(* CODESYS project Sample20190212.project

Project tree, tasks and I/O mapping:
  Device : Changsha-Cyber-MI-linux, Changsha Cyber-MI Co., Ltd., version 3.5.10.40
    application Application
      libraries: Standard, * (System); CANbus, 3.5.7.0 (3S - Smart Software Solutions GmbH); SysMem, 3.5.12.0 (System); CAA SerialCom, 3.5.12.0 (CAA Technical Workgroup); CAA Net Base Services, 3.5.12.0 (CAA Technical Workgroup); cyber gpio, 3.5.10.40 (cyber); cyber udp lib , 3.5.10.41 (cyber Inc.); SysTypes2 Interfaces, 3.5.4.0 (System); SysFile, 3.5.9.0 (System); VisuDialogs, * (System)
      task MainTask (cyclic, interval 4 ms, priority 1) calls prg_running
      task Task_running (cyclic, interval 10 ms, priority 1) calls prg_button
      task Task_CAN0 (cyclic, interval 50 ms, priority 1) calls prg_can0
      task Task_RS485 (cyclic, interval 50 ms, priority 1) calls COM_SERIAL
      task Task_Ethernet (cyclic, interval t#20ms, priority 1) calls Ethernet
      task Task_falsecheck (cyclic, interval t#20ms, priority 1) calls FaultCheck
      task Task_GPRS (cyclic, interval t#20ms, priority 1) calls GPRS
      task Task_files (cyclic, interval t#20ms, priority 1) calls Files
      task VISU_TASK (cyclic, interval 100 ms, priority 31) calls VisuElems.Visu_Prg
      CAN0/
        program prg_can0 [ST]
        function CAN_Send_MSG [ST]
      DI_DO/
        program prg_running [ST]
        program prg_button [ST]
      global variables GVL
      RS485/
        program COM_SERIAL [ST]
      Ethernet/
        data type STATE
        program Ethernet [ST]
      FaultCheck/
        function block FB_Fault [ST]
        program FaultCheck [ST]
      GPRS/
        program GPRS [ST]
      Files/
        program Files [ST]
      visualisation Visualization_files
    SoftMotion General Axis Pool
    IoDrvMIC7001 : IoDrvMIC7001, MyCompany, version 18.11.1
        input  Application.GVL.DI_button : BOOL  // Di02-Ai02@C17
        output Application.GVL.DO_running : BOOL  // LED_run
        output Application.GVL.DO_error : BOOL  // LED_err
        unmapped channels: Ai00@C16, Ai01@C28, Ai02@C17, Ai03@C29, Ai04@C30, Ai05@C19, Ai06@C31, Ai07@C20, Ai08@C18, Ai09@D18, Ai10@D20, Ai11@D31, Ai12@D19, Ai13@D30, Ai14@D29, Ai15@D17, Ai16@D28, Ai17@D16, Ai18-Do00@C25, Ai19-Do01@C24, Ai20-Do02@C13, Ai21-Do03@C01, Ai22-Do04@C03, Ai23-Do05@C04, Ai24-Do06@C05, Ai25-Do07@C06, Ai26-Do08@C08, Ai27-Do09@C09, Ai28-Do10@C10, Ai29-Do11@C11, Ai30-Do12@D34, Ai31-Do13@D35, Ai32-Do14@D23, Ai33-Do15@D12, Ai34-Do16@D10, Ai35-Do17@D09, Ai36-Do18@D08, Ai37-Do19@D07, Ai38-Do20@D05, Ai39-Do21@D04,
          Ai40-Do22@D03, Ai41-Do23@D02, Ai42-Do24@C23, Ai43-Do25@C35, Ai44-Do26@D24, Ai45-Do27@D13, Ai46-Ao00@C22, Ai47-Ao01@D14, Ai48_Pi02, Ai49_Out5V, Ai50_VCC, Ai51_VCC_L, Ai52_VCC_R, Ai53_Pwm-i0, Ai54_Pwm-i1, Ai55_Pwm-i2, Ai56_Pwm-i3, Ai57_CPU-T, Ai58_G-x, Ai59_G-y, Ai60_G-z, Ai61-reserved, Ai62-IO-cntr, Ai63-CDS-cntr, Di00-Ai00@C16, Di01-Ai01@C28, Di03-Ai03@C29, Di04-Ai04@C30, Di05-Ai05@C19, Di06-Ai06@C31, Di07-Ai07@C20, Di08-Ai08@C18, Di09-Ai09@D18, Di10-Ai10@D20, Di11-Ai11@D31, Di12-Ai12@D19, Di13-Ai13@D30, Di14-Ai14@D29, Di15-Ai15@D17, Di16-Ai16@D28,
          Di17-Ai17@D16, Di18-Ai18@C25, Di19-Ai19@C24, Di20-Ai20@C13, Di21-Ai21@C01, Di22-Ai22@C03, Di23-Ai23@C04, Di24-Ai24@C05, Di25-Ai25@C06, Di26-Ai26@C08, Di27-Ai27@C09, Di28-Ai28@C10, Di29-Ai29@C11, Di30-Ai30@D34, Di31-Ai31@D35, Di32-Ai32@D23, Di33-Ai33@D12, Di34-Ai34@D10, Di35-Ai35@D09, Di36-Ai36@D08, Di37-Ai37@D07, Di38-Ai38@D05, Di39-Ai39@D04, Di40-Ai40@D03, Di41-Ai41@D02, Di42-Ai42@C23, Di43-Ai43@C35, Di44-Ai44@D24, Di45-Ai45@D13, Di46-Ai46@C22, Di47-Ai47@D14, Di48-Pi00@C15, Di49-Pi01@C14, Di50-Pi02@D22, Di51-Pi03@D21, Di52-reserved, Di53-reserved, Di54-reserved, Di55-reserved, Di56-reserved,
          Di57-reserved, Di58-reserved, Di59-reserved, Di60-reserved, Di61-reserved, Di62-reserved, Di63-reserved, Pi00-Di48@C15, Pi01-Di49@C14, Pi02-Di50@D22, Pi03-Di51@D21, Do00-Ai18@C25, Do01-Ai19@C24, Do02-Ai20@C13, Do03-Ai21@C01, Do04-Ai22@C03, Do05-Ai23@C04, Do06-Ai24@C05, Do07-Ai25@C06, Do08-Ai26@C08, Do09-Ai27@C09, Do10-Ai28@C10, Do11-Ai29@C11, Do12-Ai30@D34, Do13-Ai31@D35, Do14-Ai32@D23, Do15-Ai33@D12, Do16-Ai34@D10, Do17-Ai35@D09, Do18-Ai36@D08, Do19-Ai37@D07, Do20-Ai38@D05, Do21-Ai39@D04, Do22-Ai40@D03, Do23-Ai41@D02, Do24-Ai42@C23, Do25-Ai43@C35, Do26-Ai44@D24, Do27-Ai45@D13, Do28-Pwmi00@C33,
          Do29-Pwmi01@C34, Do30-Pwmi02@D25, Do31-Pwmi03@D26, PWM00@C25, PWM01@C24, PWM02@C13, PWM03@C01, PWM04@C03, PWM05@C04, PWM06@C05, PWM07@C06, PWM08@C08, PWM09@C09, PWM10@C10, PWM11@C11, PWM12@D34, PWM13@D35, PWM14@D23, PWM15@D12, PWM16@D10, PWM17@D09, PWM18@D08, PWM19@D07, PWM20@D05, PWM21@D04, PWM22@D03, PWM23@D02, PWM24@C23, PWM25@C35, PWM26@D24, PWM27@D13, PWM28-Pwmi00@C33, PWM29-Pwmi01@C34, PWM30-Pwmi02@D25, PWM31-Pwmi03@D26, PWM_I_0@C33, PWM_I_1@C34, PWM_I_2@D25, PWM_I_3@D26, Ao00-Ai46@C22,
          Ao01-Ai47@D14, LED_usr, ctrl_ai_raw, ctrl_adjust, ctrl_adj0, ctrl_adj1, ctrl_adj2, ctrl_adj3, ctrl_adj4
  text list GlobalTextList
*)

// Device/Application/Ethernet/STATE
{attribute 'qualified_only'}
{attribute 'strict'}
TYPE STATE :
(
	INIT := 0, 	(* first State. Connections are set up *)
	SEND,		(* Send messages *)
	READ,		(* Receive messages *)
	ERROR		(* Prepare to reset connections *)
);
END_TYPE

// Device/Application/GVL
{attribute 'qualified_only'}
VAR_GLOBAL
	DI_button:BOOL;
	DO_running:BOOL;
	DO_error:BOOL;
END_VAR

// Device/Application/DI_DO/prg_running
PROGRAM prg_running
VAR
	cntr:DWORD:=0;
END_VAR

cntr:=cntr+1;
IF cntr<50 THEN
	gvl.DO_running:=1;	//500ms
ELSIF cntr<100 THEN
	gvl.DO_running:=0;	//1000ms
ELSE
	cntr:=0;	//开始下一个周期
END_IF

END_PROGRAM

// Device/Application/DI_DO/prg_button
PROGRAM prg_button
VAR
END_VAR

gvl.DO_error:=gvl.DI_button;

END_PROGRAM

// Device/Application/CAN0/prg_can0
PROGRAM prg_can0
VAR
	can_stat : DINT := 0;
	hCan0:CAA.HANDLE:=0;
	Err:CAA.ERROR;
	hReceiver_ready:CAA.HANDLE;
	nReceived : CAA.COUNT;
	ReadErr   : CAA.ERROR;
	nAvailable: CAA.COUNT;
	hMsg : CAA.HANDLE;
	pRxData :POINTER TO CL2I.DATA;
	tmp_byte:BYTE;
	can_data_ready:BOOL := FALSE;
	CanWriteData : ARRAY[0..7] OF BYTE;
END_VAR

CASE can_stat OF
	0:   //init can port0   
		 //初始化CAN0口
		hCan0 := cl2.DriverOpenH(usiNetId:=0,uiBaudRate:=250,xSupport29Bits:=TRUE,ctMessages:=100,peError:=ADR(Err));	 //CAN0
		IF hCan0 > 0 THEN
			can_stat := 10;
		END_IF
	
	10: //create receiver for data
		//创建接收信息的接收器: ID:0x18c21726
	  	hReceiver_ready := CL2.CreateMaskReceiver(hDriver := hCan0,
			cobIdValue := 16#18C21726, //cobID value
			cobIdMask := 16#FFFFFFFF, //cobID mask ==> all bits of value are relevant									
			xRTRValue := FALSE, //no RTR messages
			xRTRMask := FALSE, //activate RTR filter ==> xRTRValue will be checked
			x29BitIdValue := TRUE, //29 bit CAN messages
			x29BitIdMask := TRUE, //activate 29 bit filter ==> x29BitIdValue will be checked
			xTransmitValue := FALSE, //only receive messages, no transmit message loopback
			xTransmitMask := FALSE, //activate transmit mask filter ==> xTransmitValue will be checked
			xAlwaysNewest := FALSE, //FALSE := receiver with queue; TRUE: only newest message
			eEvent := CB.EVENT.NO_EVENT,  //no receive event
			xEnableSyncWindow := FALSE, //not implemented
			peError := ADR(Err) //optional pointer to error
			);
		IF (hReceiver_ready <> 0 ) THEN
			 can_stat := 20;
		ELSE
			RETURN;
		END_IF
	20:  //receive data
		//接收信息: ID:0x18c21726,  byte6.bit2  READY灯	
		nReceived := cl2.GetMsgCount(hReceiverId :=hReceiver_ready, peError := ADR(ReadErr));
		IF nReceived <> 0 THEN
			hMsg := cl2.Read(hReceiverId :=hReceiver_ready,pctMsgLeft:=ADR(nAvailable),peError:=ADR(ReadErr));
			pRxData := cl2.GetMessageDataPointer(hMessage:= hMsg,peError:=ADR(ReadErr));	
			tmp_byte := pRxData^[6];
			can_data_ready := tmp_byte.2;
			cl2.FreeMessage(hMsg);
		END_IF
		can_stat := 30;
	30:  //send data
		 //填充发送缓冲区
		CanWriteData[0] := 16#11;
		CanWriteData[1] := 16#22;
		CanWriteData[2] := 16#33;
		//发送数据
		CAN_Send_MSG(hCan0, 16#11223344, 8, CanWriteData);			
		can_stat := 20;

	100:   //error
		
END_CASE

END_PROGRAM

// Device/Application/CAN0/CAN_Send_MSG
FUNCTION CAN_Send_MSG : BOOL
VAR_INPUT
	h:	dword;     //hCan
	TMsgID   : CL2I.COBID;
    TusiLen  : USINT;
	TData    : ARRAY[0..7] OF BYTE;    	
END_VAR
VAR
   Send:CAA.HANDLE;
   WriteErr   : CL2.ERROR;
   p_data:POINTER TO CL2I.DATA;
END_VAR

IF  (0=h) THEN
	RETURN;
END_IF 

Send := cl2.CreateMessage(hDriver := h,
                          cobID := TMsgID,
						  usiLength := TusiLen,
						  xRTR := FALSE,
						  x29BitID := TRUE,
						  peError := ADR(WriteErr));
						  
IF Send <> CAA.gc_hINVALID THEN
	p_data := cl2.GetMessageDataPointer(hMessage := Send,peError:=ADR(WriteErr));
	IF (WriteErr = CL2.ERROR.NO_ERROR) THEN
		SysMemCpy(pDest:=p_data,pSrc:=ADR(TData),udiCount:=SIZEOF(TData));
	END_IF
	
	WriteErr := cl2.Write(hDriver := h,hMessage:=Send,usiPriority:=1,xEnableSyncWindow:=FALSE);
	IF (WriteErr <> CL2.ERROR.NO_ERROR) THEN
        cl2.FreeMessage(hMessage:=Send);		
	END_IF
	
	p_data := CAA.gc_pNULL;
	Send:=CAA.gc_hINVALID;	
END_IF

END_FUNCTION

// Device/Application/RS485/COM_SERIAL
PROGRAM COM_SERIAL
VAR		
	Com1Params: 			ARRAY [1..7] OF COM.PARAMETER;	(* Settings to communicate with the COM Port *)
	hCom: 					CAA.HANDLE;
	ComOpen: 				COM.Open;
	ComClose: 				COM.Close;
	ComWrite: 				COM.Write;
	ComRead: 				COM.Read;	
	
	Snd_Cnt:				CAA.SIZE;

	Rcv_Cnt: 				CAA.SIZE;
	xCom1CloseError: 		BOOL;
	xCom1WriteError: 		BOOL;
	xCom1ReadError: 		BOOL;
	xError:					BOOL;
	
	uiComState: INT := 0;
	ComID:USINT:=8;

	cmdSend:BOOL := FALSE;
	iCounter: BYTE;
	Getnumber:BYTE;
	
	Writebuffer:			ARRAY[1..14] OF BYTE;
	Readbuffer: 			ARRAY[1..16] OF BYTE;
END_VAR

CASE uiComState OF
	0:
	Com1Params[1].udiParameterId := COM.CAA_Parameter_Constants.udiPort;
	Com1Params[1].udiValue := 8;    //MIC7001的RS485接口为串口8
	Com1Params[2].udiParameterId := COM.CAA_Parameter_Constants.udiBaudrate;
	Com1Params[2].udiValue := 115200;
	Com1Params[3].udiParameterId := COM.CAA_Parameter_Constants.udiParity;
	Com1Params[3].udiValue := INT_TO_UINT(COM.PARITY.NONE);
	Com1Params[4].udiParameterId := COM.CAA_Parameter_Constants.udiStopBits;
	Com1Params[4].udiValue := INT_TO_UINT(COM.STOPBIT.ONESTOPBIT);
	Com1Params[5].udiParameterId := COM.CAA_Parameter_Constants.udiTimeout;
	Com1Params[5].udiValue := 0;
	Com1Params[6].udiParameterId := COM.CAA_Parameter_Constants.udiByteSize;
	Com1Params[6].udiValue := 8;
	Com1Params[7].udiParameterId := COM.CAA_Parameter_Constants.udiBinary;
	Com1Params[7].udiValue := 0;					
	ComOpen(xExecute := TRUE, usiListLength:=UINT_TO_USINT(SIZEOF(Com1Params)/SIZEOF(COM.PARAMETER)),pParameterList:= ADR(Com1Params),hCom=> hCom);			
	IF ComOpen.xError THEN
		uiComState := 32767;
	ELSIF ComOpen.xDone THEN
		uiComState := 1;
	END_IF
		
	
	1:
	FOR iCounter := 1 TO 14 BY 1 DO
		Writebuffer[iCounter]:=iCounter;
	END_FOR
	
	ComWrite(xExecute := TRUE,hCom:= hCom,pBuffer:= ADR(Writebuffer),szSize:= SIZEOF(Writebuffer));		
	IF ComWrite.xError THEN
		uiComState := 32767;
	END_IF
	IF ComWrite.xDone THEN		
		ComWrite(xExecute := FALSE);
		uiComState := 2;
	END_IF
	
	2:
	ComRead(xExecute := TRUE,hCom:= hCom, pBuffer:= ADR(Readbuffer), szBuffer:= SIZEOF(Readbuffer));		
	IF 	Readbuffer[1]=1 AND Readbuffer[2]=2 THEN
		Getnumber:=Readbuffer[3];
	END_IF
	IF ComRead.xError THEN
		uiComState := 32767;
	END_IF
	IF ComRead.xDone THEN
		ComRead(xExecute := FALSE);
		uiComState := 1;
	END_IF
	
	255:
	
	
	32767:	
END_CASE

END_PROGRAM

// Device/Application/Ethernet/Ethernet
PROGRAM Ethernet
VAR
	eSTATE			: STATE; (* 状态转换变量 *)
	
	myIP		: NBS.IP_ADDR; (* MIC7001本身的IP地址 *)
	myPort		: UINT; (* MIC7001用于通信的端口 *)
	IPSend		: NBS.IP_ADDR; (* 对方的IP地址 *)
	PortSend	: UINT; (* 对方的端口 *)

	sToSend			: STRING; (* 待发送数据 *)
	sReceived		: STRING; (* 接收数据 *)

	ctRecAnswers	: CAA.COUNT; (* No. of received messages *)
	ctSentMessage	: CAA.COUNT; (* No. of sent messages *)
	ctErrorCounter	: CAA.COUNT; (* No. connection errors *)

	UDPPeer			: NBS.UDP_Peer; (* FB UDP Peer *)
	UDPSend			: NBS.UDP_Send; (* FB UDP Send *)
	UDPReceive		: NBS.UDP_Receive; (* FB UDP Receive *)
	
	Peer			: CAA.HANDLE; (* Handle to the peer connection *)
	
	/// 辅助变量 
	xSend			: BOOL;
	i				: UINT;
	sTmp1			: STRING;
	xEnable			: BOOL;
END_VAR


CASE eSTATE OF

STATE.INIT:  //初始化状态
	myIP.sAddr:= '192.168.1.253';	
	myPort:= 15666;
	
	sToSend:= 'Hello World: ';
	xEnable:= TRUE;  //用于启动最下方的第70行的UDPPeer
	// 建立连接后马上转到发送状态
	IF UDPPeer.xActive THEN 
		eSTATE:= STATE.send;
	ELSIF UDPPeer.xError THEN
		eSTATE:= STATE.ERROR;
	END_IF
		
STATE.SEND:  //发送状态
	//发送一个字符串加一个数字（100到0）
	IF UDPPeer.xActive THEN 
		xSend:= TRUE;
		IF i = 0 THEN
			i:= 100;
		END_IF
		
		
		sTmp1:= concat(STR1:= sToSend, STR2:= UINT_TO_STRING(i));
		IPSend.sAddr := '192.168.1.222';	
		PortSend := 15601;
		UDPSend(xExecute:= xSend, udiTimeOut:= 0, hPeer:= Peer, ipAddr:= IPSend, uiPort:= PortSend, szSize:= len(sTmp1), pData:= ADR(sTmp1));
		//发送成功后发送的数字减一，并转入接收状态
		IF UDPSend.xDone THEN 
			i:= i -1;				
			UDPSend(xExecute:= FALSE);	
			xSend:= FALSE;
			ctSentMessage:= ctSentMessage +1;
		
			eSTATE:= STATE.read;
		ELSIF UDPSend.xError THEN
			eSTATE:= STATE.ERROR;		
		END_IF
	ELSE
		eSTATE:= STATE.ERROR;
	END_IF
	

STATE.READ:  //接收状态
	//如果收到数据，则转入发送状态，发送下一帧
	//如果出现错误，进入错误状态
	IF UDPPeer.xActive THEN 
		sReceived := '';
		UDPReceive(xEnable:= TRUE,  hPeer:= Peer, szSize:= SIZEOF(sReceived), pData:= ADR(sReceived));
		IF UDPReceive.xReady THEN
			ctRecAnswers:= ctRecAnswers +1;
			eSTATE:= STATE.SEND;
		ELSIF UDPReceive.xError THEN
			eSTATE:= STATE.ERROR;
		END_IF
	ELSE
		eSTATE:= STATE.ERROR;
	END_IF
	
STATE.ERROR:  //错误状态
	ctErrorCounter:= ctErrorCounter +1;
	xEnable := FALSE;
	eState := STATE.INIT;	 //回到初始化状态，重新开始

END_CASE

//保持每个周期调用，维护与对方的连接关系本地端口的接收状态
UDPPeer(xEnable:= xEnable, ipAddr:= myIP, uiPort:= myPort, hPeer=> Peer);

END_PROGRAM

// Device/Application/FaultCheck/FaultCheck
PROGRAM FaultCheck
VAR
	do_00:BOOL;  //do-00, 需绑定到对应的IO端口
	ai_18:DWORD; //ai-18, 需绑定到对应的IO端口
	
	do_fault_00 :FB_Fault;  //创建故障诊断功能块的实例，每个DO端口创建一个
	do_01_short_flag :BOOL := FALSE;  //短路标志
	do_01_open_flag :BOOL := FALSE;   //开路标志	
END_VAR

do_fault_00(enable := TRUE,dout := do_00, ai := ai_18);
do_01_short_flag := do_fault_00.short;
do_01_open_flag := do_fault_00.open;

RETURN;

END_PROGRAM

// Device/Application/FaultCheck/FB_Fault
FUNCTION_BLOCK FB_Fault	//检测MIC7000系列控制器高有效输出端口的短路和短线故障 功能块
VAR_INPUT
	enable :BOOL;   //开关，true 表示启用本功能块
	dout:BOOL;     	//需要检测的高有效开关量输出端口值
	ai:DWORD;      	//需要检测的高有效输出端口对应的模拟量输入值
END_VAR
VAR_OUTPUT
	ok:BOOL;    	//正常标志，为true表示无故障
	short:BOOL;  	//短路故障标志
	open:BOOL;    	//短线故障标志
END_VAR
VAR
	stat: DWORD := 0;
	stat_short :DWORD := 0;
	stat_open :DWORD := 0;
	short_cntr :DWORD := 0;
	open_cntr :DWORD := 0;
END_VAR
VAR CONSTANT   //参数定义，可以根据情况修改
	SHORT_VALUE :DWORD := 3000; //短路门槛值
	OPEN_VALUE :DWORD := 25;   	//开路门槛值
	TIME_OUT :DWORD := 10;   	//超时周期数
END_VAR

IF NOT enable THEN
	ok := TRUE;
	short := FALSE;
	open := FALSE;
	short_cntr := 0;
	open_cntr := 0;
	RETURN;
END_IF

CASE stat OF
	0:
		ok := TRUE;
		short := FALSE;
		open := FALSE;
		IF dout THEN  
			stat := 100;	// dout high, detect short
			stat_short := 0;
		ELSE 
			stat := 200;  //dout low, detect open
			stat_open := 0;
		END_IF
	
	100:  //detect short
		IF NOT dout THEN  //return 
			stat := 0;
		END_IF
		CASE stat_short OF
			0:
				short := FALSE;
				IF ai < SHORT_VALUE THEN  //short
					stat_short := 10;
					short_cntr := 0;
				END_IF
			10:  //short wait for timeout
				IF ai > SHORT_VALUE THEN  //normal , wait for return
					IF short_cntr = 0 THEN
						stat_short := 0;
					ELSE
						short_cntr := short_cntr - 1;
					END_IF
				ELSE  //short, 
					IF short_cntr > TIME_OUT THEN
						short := TRUE;
					ELSE
						short_cntr := short_cntr + 1;
					END_IF		
				END_IF	
		END_CASE

	200:
		IF dout THEN  //  dout high, return to detect short
			stat := 0;
		END_IF
		CASE stat_open OF
			0:
				open := FALSE;
				IF ai > OPEN_VALUE THEN  //open
					stat_open := 10;
					open_cntr := 0;
				END_IF
			10:
				IF ai < OPEN_VALUE THEN  //normal, wait for return
					IF open_cntr = 0 THEN
						stat_open := 0;
					ELSE
						open_cntr := open_cntr - 1;
					END_IF
				ELSE
					IF open_cntr > TIME_OUT THEN
						open := TRUE;
					ELSE
						open_cntr := open_cntr + 1;
					END_IF
				END_IF			
		END_CASE
END_CASE

ok := (NOT short) AND (NOT open);

END_FUNCTION_BLOCK

// Device/Application/GPRS/GPRS
PROGRAM GPRS
VAR
	is_inited :BOOL := FALSE;
	
	udp_handle :CAA.HANDLE; 
	udp_init_fb:Udp_Init;
	udp_write_fb:Udp_Write;
	udp_read_fb:Udp_Read;

	Writebuffer: 			ARRAY[1..200] OF BYTE;
	Readbuffer: 			ARRAY[0..1499] OF BYTE;
	
	atcState :INT := 0;
	ton_fb :TON;
	
END_VAR


IF NOT is_inited THEN
	udp_init_fb(ip_addr := '47.107.240.29', port := 34567);
	IF udp_init_fb.init_mode = 1 THEN
		is_inited := TRUE;
		udp_handle := udp_init_fb.udp_handle;
		atcState := 0;
		Writebuffer[1] := 0;
		Writebuffer[2] := 1;
		Writebuffer[3] := 2;
		Writebuffer[4] := 3;
		Writebuffer[5] := 4;
		Writebuffer[6] := 5;
		Writebuffer[7] := 6;
		Writebuffer[8] := 7;
		Writebuffer[9] := 8;
		Writebuffer[10] := 9;
		Writebuffer[11] := 10;
		Writebuffer[12] := 11;
		Writebuffer[13] := 12;
		Writebuffer[14] := 13;
		Writebuffer[15] := 14;
		Writebuffer[16] := 15;
		Writebuffer[17] := 16;
		Writebuffer[18] := 17;
		Writebuffer[19] := 18;
		Writebuffer[20] := 19;
		Writebuffer[21] := 20;
	END_IF
END_IF


IF is_inited = TRUE THEN
	CASE atcState OF
	0:  //发送数据
		// if error, atcState return 32767, if done, atcState return 1
		//GPRS网络读取和发送数据是否成功通过atcState是否为255判断，等于255表示成功，不等于255表示不成功
	udp_write_fb(com := udp_handle, buffer:= ADR(Writebuffer), size := 21);
	(*
	IF udp_write_fb.atcState = 255 THEN
		atcState := 2;
	END_IF	
	*)
	atcState := 2;
	
	2:
	ton_fb(IN := TRUE, PT := TIME#3000MS);
	IF (ton_fb.Q) THEN
		ton_fb(IN := FALSE, PT := TIME#3000MS);
		atcState := 3;
	END_IF	
		
	3:
	udp_read_fb(com:= udp_handle, buffer:= ADR(Readbuffer), rsize := SIZEOF(Readbuffer));
	(*	
	IF udp_read_fb.atcState = 255 THEN
		atcState := 0;
	END_IF
	*)
	atcState := 0;
	END_CASE	
END_IF

END_PROGRAM

// Device/Application/Files/Files
PROGRAM Files
VAR
	hFile: RTS_IEC_HANDLE;
	udiOpenError: RTS_IEC_RESULT;
	udiReadError: RTS_IEC_RESULT;
		
	WriteEnable: BOOL;
	para_val:STRING(256); 	
	data1: BYTE;
	data2: BYTE;
	data3: BYTE;
	data4: BYTE;
	data5: BYTE;
	data6: BYTE;
	udiByteWrite: __XWORD;
	udiWriteError: RTS_IEC_RESULT;
	ReadEnable: BOOL;
	udiPos: UDINT;
	udiByteRead: UDINT;
	str: STRING(256);
	data1_read: BYTE;
	data2_read: BYTE;
	data3_read: BYTE;
	data4_read: BYTE;
	data5_read: BYTE;
	data6_read: BYTE;
END_VAR
VAR CONSTANT
	para_file:STRING:=ANY_TO_STRING("parameters.txt");
END_VAR

//写文件
IF WriteEnable THEN
	para_val[0] := data1;
	para_val[1] := data2;
	para_val[2] := data3;
	para_val[3] := data4;
	para_val[4] := data5;
	para_val[5] := data6;
	
	hFile := sysfileopen(szFile := para_file, am := sysfile.AM_WRITE, pResult:= ADR(udiOpenError));
	IF hFile = RTS_INVALID_HANDLE	THEN  //文件不存在
		WriteEnable:=FALSE;
		RETURN;
	END_IF
	udiByteWrite := sysfile.SysFileWrite(hFile := hFile,pbyBuffer := ADR(para_val),ulSize := ANY_TO_DWORD(len(para_val)), pResult := ADR(udiWriteError));
	sysfile.SysFileClose(hFile);
	//WriteEnable:=FALSE;
END_IF

//读文件
IF ReadEnable THEN
	hFile := sysfileopen(szFile := para_file, am := sysfile.AM_READ, pResult:= ADR(udiOpenError));
	IF hFile = RTS_INVALID_HANDLE	THEN  //文件不存在
		ReadEnable:=FALSE;
		RETURN;
	END_IF
	
	udiPos := SysFileSetPos(hFile:=hFile, ulOffset := 0);	
	udiByteRead := sysfile.SysFileRead(hfile := hFile,pbyBuffer := ADR(str), ulSize := SIZEOF(str), pResult := ADR(udiReadError));
	data1_read:=str[0];
	data2_read:=str[1];
	data3_read:=str[2];
	data4_read:=str[3];
	data5_read:=str[4];
	data6_read:=str[5];
	sysfile.SysFileClose(hFile);
	//ReadEnable:=FALSE;
END_IF

END_PROGRAM

// Device/Application/Visualization_files
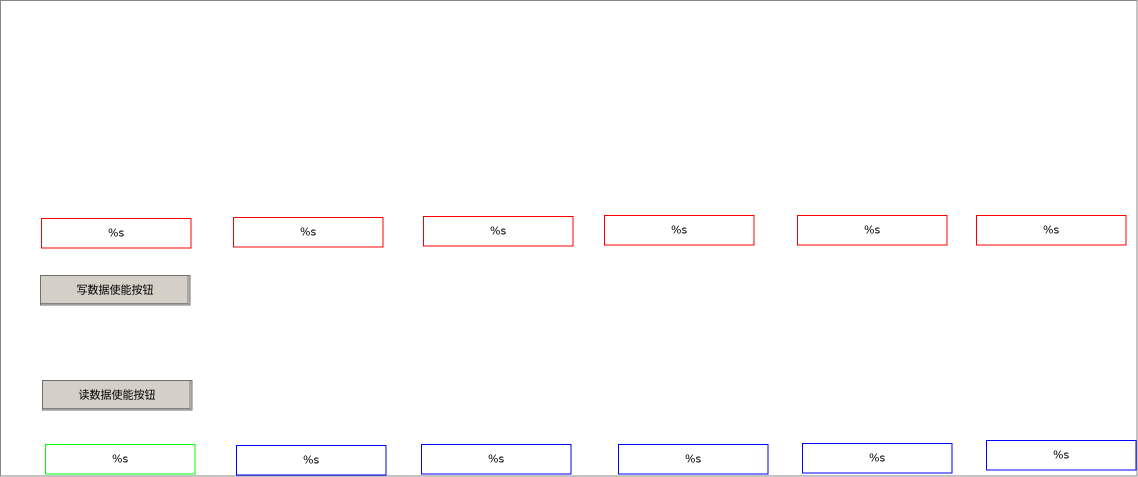
VISUALIZATION Visualization_files  // 1138x477
    Button (40,275 150x30), "写数据使能按钮"
        OnMouseLeave: execute { Files.WriteEnable:=false; }
        OnMouseClick: execute { Files.WriteEnable:=true; }
    Textfield (41,218 150x30), "%s", text variable: Files.data1
        OnMouseEnter: write Files.data1 via Default
    Textfield (423,216 150x30), "%s", text variable: Files.data3
        OnMouseEnter: write Files.data3 via Default
    Textfield (797,215 150x30), "%s", text variable: Files.data5
        OnMouseEnter: write Files.data5 via Default
    Button (42,380 150x30), "读数据使能按钮"
        OnMouseLeave: execute { Files.ReadEnable:=false; }
        OnMouseClick: execute { Files.ReadEnable:=true; }
    Textfield (236,445 150x30), "%s", text variable: Files.data2_read
    Textfield (421,444 150x30), "%s", text variable: Files.data3_read
    Textfield (618,444 150x30), "%s", text variable: Files.data4_read
    Textfield (802,443 150x30), "%s", text variable: Files.data5_read
    Textfield (986,440 150x30), "%s", text variable: Files.data6_read
    Textfield (233,217 150x30), "%s", text variable: Files.data2
        OnMouseEnter: write Files.data2 via Default
    Textfield (604,215 150x30), "%s", text variable: Files.data4
        OnMouseEnter: write Files.data4 via Default
    Textfield (976,215 150x30), "%s", text variable: Files.data6
        OnMouseEnter: write Files.data6 via Default
    Textfield (45,444 150x30), "%s", text variable: Files.data1_read
END_VISUALIZATION
